FUNCTION_BLOCK FB_MotionAxisMoveAbsoluteNC IMPLEMENTS I_MotionAxisMoveAbsolute
VAR
END_VAR

END_FUNCTION_BLOCK

(* stored: Version 1.1.0.1
   POU FB_MotionAxisMoveAbsoluteNC: Id {97842839-d991-4d0e-9427-5c5a6246ff33}, SpecialFunc None *)
